FUNCTION Convert_SINT_TO_BOOL : Hresult
VAR_INPUT
	in : SINT;
	out : REFERENCE TO BOOL;
END_VAR
VAR
	converted : BOOL;
END_VAR
VAR CONSTANT
	INCOMPATIBLE : HRESULT := 16#9811070E;
END_VAR

converted := SINT_TO_BOOL(in);

IF (BOOL_TO_SINT(converted) <> in) THEN
	Convert_SINT_TO_BOOL := INCOMPATIBLE;
	RETURN;
END_IF

out := converted;

END_FUNCTION

(* stored: Version 1.1.0.1, ProductVersion 3.1.4024.12
   POU Convert_SINT_TO_BOOL: Id {fe711f65-df05-4817-ab71-eb70c153fbe9}, SpecialFunc None *)
